FUNCTION_BLOCK FB_DancerCtrl
VAR_INPUT
	Enable	: BOOL;
	DancerFull:BOOL;
	DancerPosition	:REAL;
	Ctrl_Type	: E_DancerCtrlTyp;
	//Ctrl_ref:				REFERENCE TO Ctrl_Typ;
END_VAR
VAR_OUTPUT
	Jog:BOOL;
	dancerFullStatus:BOOL;
END_VAR
VAR
	FilterOn:TON:=(PT:=T#50MS);
	FilterOff:TON:=(PT:=T#50MS);
	
	PositionMax	: REAL := 200;//mm
	PositionMin	: REAL := 100;//mm
END_VAR


IF Enable THEN
	
	IF Ctrl_Type = E_DancerCtrlTyp.DIGITAL THEN
		ACT_Digital();
	ELSIF Ctrl_Type = E_DancerCtrlTyp.ANALOG	THEN
		ACT_Analog();
	END_IF

ELSE
	Jog := FALSE;
	dancerFullStatus := FALSE;
END_IF

ACTION ACT_Analog:


IF DancerPosition > PositionMax THEN
	Jog := TRUE;
ELSIF
	DancerPosition < PositionMin THEN
	 Jog := FALSE;	
END_IF

 dancerFullStatus := (DancerPosition < PositionMax);
END_ACTION

ACTION ACT_Digital:


	FilterOn(IN:=DancerFull);
	FilterOff(IN:=NOT(DancerFull));

	IF (DancerFull  = TRUE) AND FilterOn.Q  THEN
		Jog:=FALSE;
	ELSIF FilterOff.Q THEN
		Jog:=TRUE;
	END_IF
	
dancerFullStatus := FilterOn.Q;
END_ACTION

END_FUNCTION_BLOCK

(* stored: Version 1.1.0.1, ProductVersion 3.1.4024.3
   POU FB_DancerCtrl: Id {33976128-a633-4b6c-8520-3f52b4a5b0f8}, SpecialFunc None
   Action ACT_Analog: Id {0b6be42d-08fe-483f-9b32-d82c11e3b756}
   Action ACT_Digital: Id {589b2d82-991e-44fb-83dd-c60e7de41b5d} *)
